TYPE
    ST_AssemblyEnd : STRUCT
        SeqID : UDINT;
    END_STRUCT
END_TYPE

(* stored: Version 1.1.0.1
   DUT ST_AssemblyEnd: Id {fcc54c7e-1c2d-40ce-a825-5ea4a7590304} *)
